(* CoDeSys 2.3 export: TEPLOTA.EXP *)

(* POU teplota, FBD *)
PROGRAM teplota
VAR
	tempF: WORD;
	tempC: WORD;
	chooseTemp: RS;
	trigC: R_TRIG;
	trigF: R_TRIG;
	test: WORD;
	select: BOOL;
	count: counter;
	tempSet: WORD;
	stykacSet: RS;
	tempOut: WORD;
	pickDisp: RS;
	dispOut: WORD;
	pickUnit: RS;
	pickDispSR: SR;

	hu:BOOL:=FALSE;
	hl:BOOL:=TRUE;

	hysterezeSet:BYTE:=2;
	hystereze:WORD;

	check: WORD;
END_VAR
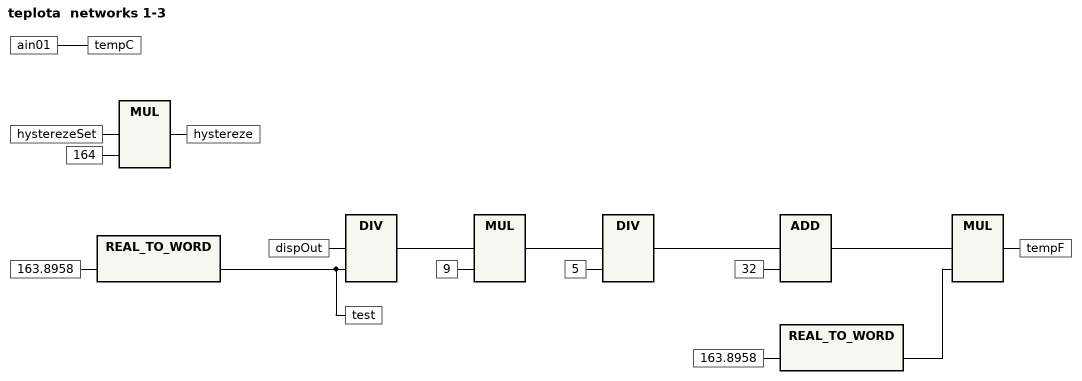
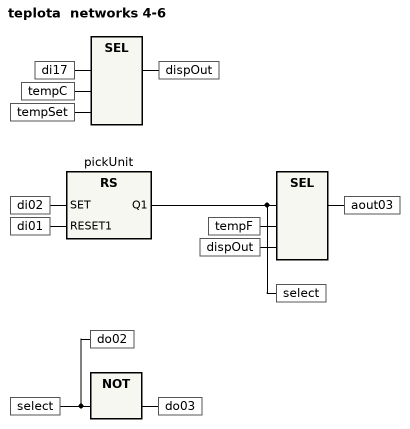
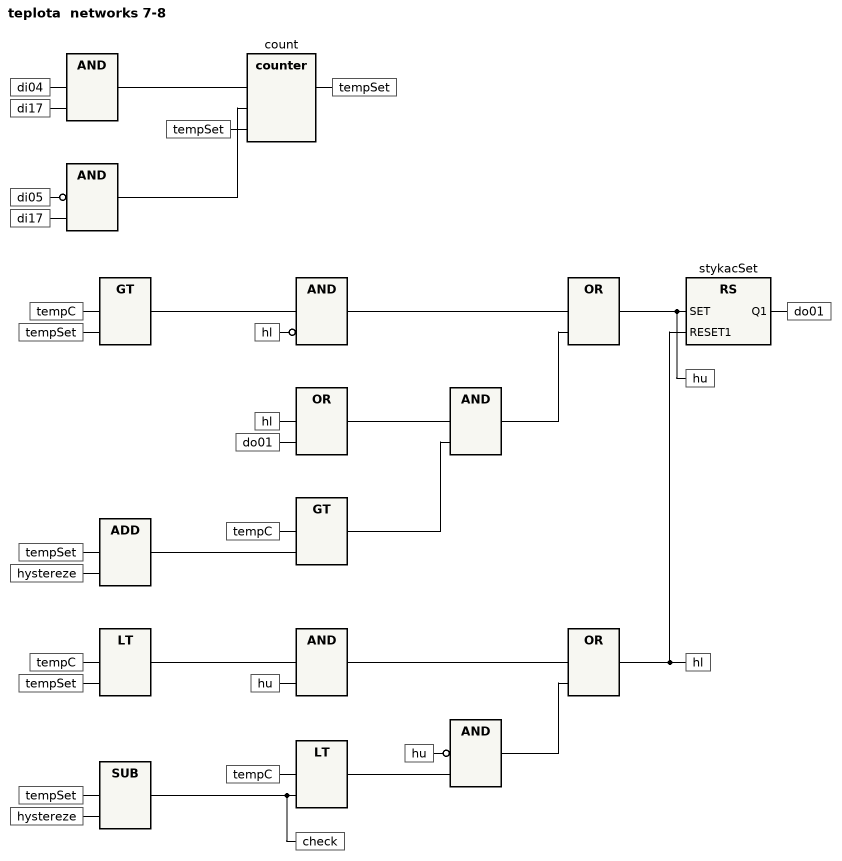
_FBD_ (* Function Block Diagram *)
NETWORK 1 (*prevedeni hodnoty teplomeru na promennou tempC*):
	ain01 => tempC
NETWORK 2
	MUL(hysterezeSet, 164) => hystereze
NETWORK 3 (*prevod hodnoty displaye na Fahrenheit*):
	MUL(ADD(DIV(MUL(DIV(dispOut, <REAL_TO_WORD(163.8958) => test>), 9), 5), 32), REAL_TO_WORD(163.8958)) => tempF
NETWORK 4
	SEL(di17, tempC, tempSet) => dispOut
NETWORK 5
	SEL(<pickUnit:RS(SET: di02, RESET1: di01) => select>, tempF, dispOut) => aout03
NETWORK 6 (*vyber ledky*):
	NOT(<select => do02>) => do03
NETWORK 7 (*nastaveni hodnoty teplomeru*):
	count:counter(AND(di04, di17), AND(NOT di05, di17), tempSet) => tempSet
NETWORK 8 (*porovnani hodnot a spinani vystupu accordingly*):
	stykacSet:RS(SET: <OR(AND(GT(tempC, tempSet), NOT hl), AND(OR(hl, do01), GT(tempC, ADD(tempSet, hystereze)))) => hu>, RESET1: <OR(AND(LT(tempC, tempSet), hu), AND(NOT hu, LT(tempC, <SUB(tempSet, hystereze) => check>))) => hl>) => do01
_END_FBD_
(* the same logic as Structured Text *)
(* Network 1: see the listing above *)
(* Network 2 *)
hystereze := hysterezeSet * 164;
(* Network 3: see the listing above *)
(* Network 4 *)
dispOut := SEL(di17, tempC, tempSet);
(* Network 5 *)
pickUnit(SET := di02, RESET1 := di01);
select := pickUnit.Q1;
aout03 := SEL(pickUnit.Q1, tempF, dispOut);
(* Network 6: see the listing above *)
(* Network 7: see the listing above *)
(* Network 8: see the listing above *)
END_PROGRAM
